PROGRAM tcp_ip
VAR
	createConn: BOOL;
	FB_create : FB_SocketListen;
	
	data: ARRAY[0..5000] OF BYTE;
	
END_VAR

FB_create(
sSrvNetId := '',
sLocalHost := '127.0.0.1',
nLocalPort := 811,
tTimeout := DEFAULT_ADS_TIMEOUT
);

END_PROGRAM

(* stored: Version 1.1.0.1, ProductVersion 3.1.4024.0
   POU tcp_ip: Id {de64ce75-9f89-4066-b8fa-6c9812ac26d8}, SpecialFunc None *)
